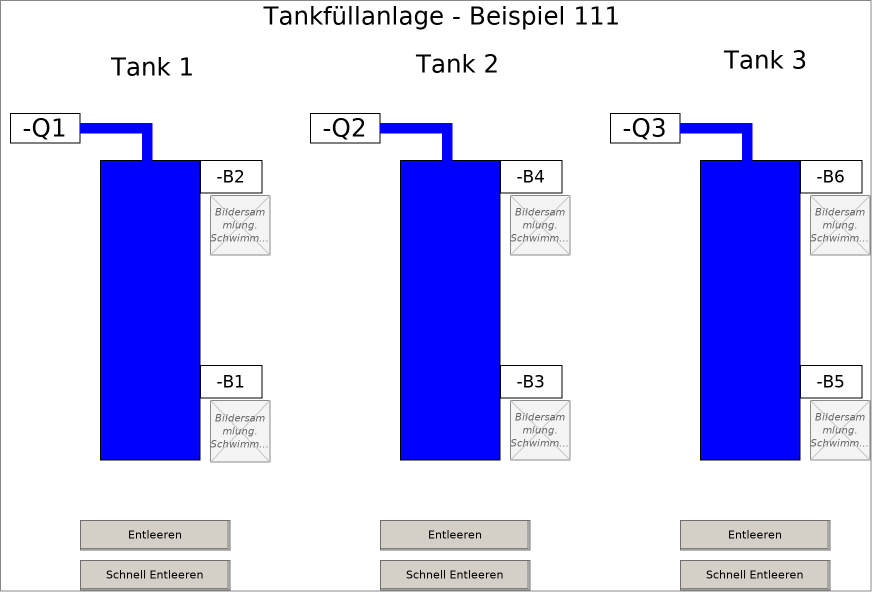
VISUALIZATION TankFuellAnlage  // 872x592
    Polygon (680,123) (752,123) (753,459) (743,459) (742,133) (680,133)
    Polygon (380,123) (452,123) (453,459) (443,459) (442,133) (380,133)
    Polygon (80,123) (152,123) (153,459) (143,459) (142,133) (80,133)
    Rectangle (100,160 100x300)
    Rectangle (100,160 100x300)
        p2773130477: MAIN.DigitalTwin.uiFuellstandTank1
    Label (105,52 95x30), "Tank 1"
    Button (80,520 150x30), "Entleeren"
        tap MAIN.DigitalTwin.xAuslass1
    Rectangle (10,113 70x30), "-Q1", colour toggle: DIO.Ventil_1
    Rectangle (400,160 100x300)
    Rectangle (400,160 100x300)
        p2773130477: MAIN.DigitalTwin.uiFuellstandTank2
    Label (410,49 95x30), "Tank 2"
    Button (380,520 150x30), "Entleeren"
        tap MAIN.DigitalTwin.xAuslass2
    Rectangle (310,113 70x30), "-Q2", colour toggle: DIO.Ventil_2
    Rectangle (391,183 29x301), colour toggle: DIO.Ventil_1
    Rectangle (700,160 100x300)
    Rectangle (700,160 100x300)
        p2773130477: MAIN.DigitalTwin.uiFuellstandTank3
    Label (718,45 95x30), "Tank 3"
    Button (680,520 150x30), "Entleeren"
        tap MAIN.DigitalTwin.xAuslass3
    Rectangle (610,113 70x30), "-Q3", colour toggle: DIO.Ventil_3
    Image (810,195 50x60), invisible if: dio.Schwimmerschalter_B6, image: Bildersammlung.Schwimmerschalter_Offen
    Image (810,195 60x60), invisible if: NOT dio.Schwimmerschalter_B6, image: Bildersammlung.Schwimmerschalter_Betätigt
    Image (810,400 50x60), invisible if: dio.Schwimmerschalter_B5, image: Bildersammlung.Schwimmerschalter_Offen
    Image (510,195 50x60), invisible if: dio.Schwimmerschalter_B4, image: Bildersammlung.Schwimmerschalter_Offen
    Image (510,400 50x60), invisible if: dio.Schwimmerschalter_B3, image: Bildersammlung.Schwimmerschalter_Offen
    Image (210,195 50x60), invisible if: dio.Schwimmerschalter_B2, image: Bildersammlung.Schwimmerschalter_Offen
    Image (210,400 50x60), invisible if: dio.Schwimmerschalter_B1, image: Bildersammlung.Schwimmerschalter_Offen
    Image (810,400 60x60), invisible if: NOT dio.Schwimmerschalter_B5, image: Bildersammlung.Schwimmerschalter_Betätigt
    Image (510,195 60x60), invisible if: NOT dio.Schwimmerschalter_B4, image: Bildersammlung.Schwimmerschalter_Betätigt
    Image (510,400 60x60), invisible if: NOT dio.Schwimmerschalter_B3, image: Bildersammlung.Schwimmerschalter_Betätigt
    Image (210,195 60x60), invisible if: NOT dio.Schwimmerschalter_B2, image: Bildersammlung.Schwimmerschalter_Betätigt
    Image (210,400 60x62), invisible if: NOT dio.Schwimmerschalter_B1, image: Bildersammlung.Schwimmerschalter_Betätigt
    Rectangle (500,160 62x33), "-B4"
    Rectangle (200,160 62x33), "-B2"
    Rectangle (800,160 62x33), "-B6"
    Rectangle (200,365 62x33), "-B1"
    Rectangle (500,365 62x33), "-B3"
    Rectangle (800,365 62x33), "-B5"
    Polygon (80,123) (152,123) (153,459) (143,459) (142,133) (80,133), invisible if: NOT DIO.Ventil_1
    Polygon (380,123) (452,123) (453,459) (443,459) (442,133) (380,133), invisible if: NOT DIO.Ventil_2
    Polygon (680,123) (752,123) (753,459) (743,459) (742,133) (680,133), invisible if: NOT DIO.Ventil_3
    Label (139,1 606x30), "Tankfüllanlage - Beispiel 111"
    Button (80,560 150x30), "Schnell Entleeren"
        tap MAIN.DigitalTwin.xSchnellEntleeren1
    Button (380,560 150x30), "Schnell Entleeren"
        tap MAIN.DigitalTwin.xSchnellEntleeren2
    Button (680,560 150x30), "Schnell Entleeren"
        tap MAIN.DigitalTwin.xSchnellEntleeren3
END_VISUALIZATION

(* stored: Version 1.1.0.1, ProductVersion 3.1.4022.7
   Visu TankFuellAnlage: Id {116ef40b-496c-489a-a025-1af3552c8f1e} *)
